Staubli VAL3: cumsum.pgx

public program cumsum(num& x_nInput[], num& x_nResult[])
  local num l_nLength
  local num l_nElement
begin

  l_nLength = size(x_nInput)
  x_nResult[0] = 0
  resize(x_nResult,1,l_nLength)

  for l_nElement = 0 to l_nLength-1
    if l_nElement == 0
      x_nResult[0] = x_nInput[0]
    else
      x_nResult[l_nElement] = x_nResult[l_nElement-1] + x_nInput[l_nElement]
    endIf

  endFor

end
